PROGRAM FadenzugmotorAnAus
VAR
	PowerFadenzugmotor: MC_Power;
	PowerFadenzugmotorOut: ST_McOutputs;
	ResetFadenzugmotor: MC_Reset;
	ResetFadenzugmotorOut: ST_McOutputs;
	HaltFadenzugmotor: MC_Halt;
	HaltFadenzugmotorOut: ST_McOutputs;
	HomeFadenzugmotor: MC_Home;
	HomeFadenzugmotorOut: ST_McOutputs;
	MoveAbFadenzugmotorOut1: ST_McOutputs;
	MoveAbFadenzugmotor1: MC_MoveAbsolute;
	MoveAbFadenzugmotor2: MC_MoveAbsolute;
	MoveAbFadenzugmotorOut2: ST_McOutputs;
	MC_Stop1: MC_Stop;
	MC_StopOut1: ST_McOutputs;
	HaltAufwicklerOut: ST_McOutputs;
	HaltAbwicklerOut: ST_McOutputs;
	AbwicklerMoveV_Out: ST_McOutputs;
	AufwicklerMoveV: MC_MoveVelocity;
	HaltAbwickler: MC_Halt;
	HaltAufwickler: MC_Halt;
	PowerAbwickler: MC_Power;
	PowerAbwicklerOut: ST_McOutputs;
	PowerAufwickler: MC_Power;
	PowerAufwicklerOut: ST_McOutputs;
	HomeAbwickler: MC_Home;
	HomeAbwicklerOut: ST_McOutputs;
	HomeAufwickler: MC_Home;
	HomeAufwicklerOut: ST_McOutputs;
	ResetAbwickler: MC_Reset;
	ResetAbwickleOUT: ST_McOutputs;
	ResetAufwickler: MC_Reset;
	ResetAufwickleOUT: ST_McOutputs;
	MasterMoveV: MC_MoveVelocity;
	HaltMasterachse: MC_Halt;
	ResetMasterachseOut: ST_McOutputs;
	HomeMasterachseOut: ST_McOutputs;
	HaltMasterachseOut: ST_McOutputs;
	PowerMasterachseOut: ST_McOutputs;
	GearIn_M_AB_Out: ST_McOutputs;
	MasterMoveV_Out: ST_McOutputs;
	PowerMasterachse: MC_Power;
	HomeMasterachse: MC_Home;
	ResetMasterachse: MC_Reset;
	GearIn_M_AB: MC_GearIn;
	GearOut_M_AB: MC_GearOut;
	CamIn_AB_AUF_Out: ST_McOutputs;
	GearOut_M_AB_Out: ST_McOutputs;
	CamIn_AB_AUF: MC_CamIn;
	CamOut_AB_AUF: MC_CamOut;
	JogFadenzugmotorOut: ST_McOutputs;
	CamOut_AB_AUF_Out: ST_McOutputs;
	startFadenzugTrig: R_TRIG;
	flag: INT;
	JogFadenzugmotor: MC_Jog;
	// Zustandsvariable Hauptprogramm
	stateFadenzugmotor: MoveState_Fadenzugmotor;
	
END_VAR

GlobaleVariablen.Fadenzugmotor();
IF Fadenzugmotor.NcToPlc.ActPos > 89 AND Fadenzugmotor.NcToPlc.ActPos < 91 THEN
	FadenzugHomingFertig := TRUE;
ELSE FadenzugHomingFertig := FALSE;
END_IF
IF DTD_CTD THEN
	TrackingDifferentiator(Sollkraft);
ELSE
	DiscreteTrackingDifferentiator(Sollkraft);
END_IF

ESO(Fadenzugkraft_2);

// Programmablauf mittels Zustandsautomat
CASE stateFadenzugmotor OF
(* ===========================================================================================
	Zustand 1: Programm ist im Ausgangszustand und wartet auf Benutzereingabe. Alle 
	Funktionsbausteine werden initialisiert, etwaige Fehler zurückgesetzt. *)	
	FADENZUG_INIT:
		FadenzugmotorStopp := FALSE;
		MoveAbFadenzugmotor1.Execute := FALSE;
		MoveAbFadenzugmotor2.Execute := FALSE;
		FadenzugmotorLaeuft := FALSE;
		ResetFadenzugmotor.Execute := FALSE;
		HaltFadenzugmotor.Execute := FALSE;
		FadenmotorRegeln := FALSE;
		IF FadenmotorFreigabe THEN
			stateFadenzugmotor := FADENZUG_POWER_ON;
		ELSE
			PowerFadenzugmotor.Enable := FALSE;
			PowerFadenzugmotor.Enable_Positive := FALSE;
			PowerFadenzugmotor.Enable_Negative := FALSE;
		END_IF
(* ===========================================================================================
	Zustand 2: Schlalten der allgemeinen Software-Freigabe, Vorschubfreigabe in positive Richtung
	durch MC_Power. Sobald Funktionsbaustein MC_Power die Betriebsbereitschaft der Achse signalisiert,
	Zustandsübergang in Forward*)
	FADENZUG_POWER_ON:
		IF FadenmotorFreigabe = TRUE THEN
			PowerFadenzugmotor.Enable := TRUE;
			PowerFadenzugmotor.Enable_Positive := TRUE;
			PowerFadenzugmotor.Enable_Negative := TRUE;
			FadenzugmotorStopp := FALSE;
			IF PowerFadenzugmotorOut.Done THEN
				IF FadenzugJogStart THEN
					stateFadenzugmotor := FADENZUG_JOG;
				END_IF
			ELSIF PowerFadenzugmotor.Error THEN
				stateFadenzugmotor := FADENZUG_ERROR;
			END_IF
		ELSIF FadenmotorFreigabe = FALSE THEN
			stateFadenzugmotor := FADENZUG_HALT_ZU_INT;
		END_IF
(* ===========================================================================================
	Zustand 3: Setzten der Ist-Position auf 90 Grad*)			
	FADENZUG_JOG:
		IF FadenmotorFreigabe = TRUE THEN
			FadenzugmotorJogLaeuft := TRUE;
			ActJog();
			IF FadenzugJogStart = FALSE THEN
				FadenzugmotorJogLaeuft := FALSE;
				IF FadenmotorRegeln = TRUE THEN
					stateFadenzugmotor := FADENZUG_MOVE;
				END_IF
			END_IF
		ELSIF FadenmotorFreigabe = FALSE THEN
			stateFadenzugmotor := FADENZUG_HALT_ZU_INT;
		END_IF
(* ===========================================================================================
	Zustand 4: Starten des Fadenzugmotors mithilfe der Fadenzugspannung. Zustandsübergang durch Bedienerbefehl.*)	
	FADENZUG_MOVE:
	
		IF FadenmotorFreigabe = TRUE THEN
			
			IF FadenzugmotorStopp = TRUE THEN
				FadenmotorFreigabe := FALSE;
			END_IF
			//*********Positionsführungsgröße berechnen*************
			PRG_PID_Fadenzugmotor();
			IF ILC_EinAus = TRUE AND MasterStart = TRUE THEN
				ILC();
				MoveAbFadenzugmotor1.Position := ILC_Out + GlobaleVariablen.Fadenzugmotor.NcToPlc.ActPos + _u;
			ELSE
				MoveAbFadenzugmotor1.Position := GlobaleVariablen.Fadenzugmotor.NcToPlc.ActPos + _u;
			END_IF
			
			MoveAbFadenzugmotor1.Velocity := 60000;
			ActBegrenzung_1();
			//******************************************************
			
			MoveAbFadenzugmotor1.Execute := TRUE;
			FadenzugmotorLaeuft := TRUE;
			
			//*********Zustand umschalten***************************
			IF MoveAbFadenzugmotorOut1.Busy OR MoveAbFadenzugmotorOut1.Active THEN
				MoveAbFadenzugmotor1.Execute := FALSE;
				stateFadenzugmotor := FADENZUG_MOVE_NEW;
			END_IF
			
			IF MoveAbFadenzugmotorOut1.Done OR MoveAbFadenzugmotorOut1.CommandAborted THEN
				MoveAbFadenzugmotor1.Execute := FALSE;
				stateFadenzugmotor := FADENZUG_MOVE;
			END_IF

			IF MoveAbFadenzugmotorOut1.Error THEN
				stateFadenzugmotor := FADENZUG_ERROR;
			END_IF
			//******************************************************
		ELSIF FadenmotorFreigabe = FALSE THEN
			stateFadenzugmotor := FADENZUG_HALT_ZU_INT;
		END_IF
(* ===========================================================================================		
	Zustand 5: Die Funktion ist gleich wie Zustand 4, aber mithilfe dises Zustands kann den letzte Positionsbefehel unterbrechen 
	und schnell den neue Positionsbefehel aktualisieret und ersetzt werden. *)		
	FADENZUG_MOVE_NEW:

		IF FadenmotorFreigabe = TRUE THEN
			
			IF FadenzugmotorStopp = TRUE THEN
				FadenmotorFreigabe := FALSE;
			END_IF
			
			//*********Positionsführungsgröße berechnen*************
			PRG_PID_Fadenzugmotor();
			IF ILC_EinAus = TRUE AND MasterStart = TRUE THEN
				ILC();
				MoveAbFadenzugmotor2.Position := ILC_Out + GlobaleVariablen.Fadenzugmotor.NcToPlc.ActPos + _u;
			ELSE
				MoveAbFadenzugmotor2.Position := GlobaleVariablen.Fadenzugmotor.NcToPlc.ActPos + _u;
			END_IF
			MoveAbFadenzugmotor2.Velocity := 60000;
			ActBegrenzung_2();
			//******************************************************
			
			MoveAbFadenzugmotor2.Execute := TRUE;
			FadenzugmotorLaeuft := TRUE;
			
			//*********Zustand umschalten***************************
			IF MoveAbFadenzugmotorOut2.Busy OR MoveAbFadenzugmotorOut2.Active THEN
				MoveAbFadenzugmotor2.Execute := FALSE;
				stateFadenzugmotor := FADENZUG_MOVE;
			ELSIF MoveAbFadenzugmotorOut2.Done OR MoveAbFadenzugmotorOut2.CommandAborted THEN
				MoveAbFadenzugmotor2.Execute := FALSE;
				stateFadenzugmotor := FADENZUG_MOVE_NEW;
			ELSIF MoveAbFadenzugmotorOut2.Error THEN
				stateFadenzugmotor := FADENZUG_ERROR;
			END_IF
			//******************************************************
		ELSIF FadenmotorFreigabe = FALSE THEN
			stateFadenzugmotor := FADENZUG_HALT_ZU_INT;
		END_IF
(* ===========================================================================================
   Zustand 7: Anhalten des Fadenzugmotors, im Anschluss Rückkehr in den Ausgangszustand. *)			
	FADENZUG_HALT_ZU_INT:
		MoveAbFadenzugmotor1.Execute := FALSE;
		MoveAbFadenzugmotor2.Execute := FALSE;
		HaltFadenzugmotor.Execute := TRUE;
		IF HaltFadenzugmotorOut.Done THEN
			FadenzugmotorStopp := TRUE;
			FadenmotorFreigabe := FALSE;
			FadenzugmotorLaeuft := FALSE;
			HaltFadenzugmotor.Execute := FALSE;
			stateFadenzugmotor := FADENZUG_INIT;
		ELSIF HaltFadenzugmotorOut.Error OR HaltFadenzugmotorOut.CommandAborted THEN
			HaltFadenzugmotor.Execute := FALSE;
			stateFadenzugmotor := FADENZUG_ERROR;
		END_IF

(* ===========================================================================================
   Zustand 8: Im Falle eines Bausteinfehlers wird überprüft, ob sich die Achse ebenfalls im    
   Fehlerzustand befindet, was einen Achsreset erfordert. Andernfalls werden Bausteinfehler 
   im Zustand Init zurückgesetzt.*)				
	FADENZUG_ERROR:
		MoveAbFadenzugmotor1.Execute := FALSE;
		MoveAbFadenzugmotor2.Execute := FALSE;
		PowerFadenzugmotor.Enable := FALSE;
		FadenmotorFreigabe := FALSE;
		IF Fadenzugmotor.Status.Error THEN
			stateFadenzugmotor := FADENZUG_RESET;	// Reset bei Achsfehler
		ELSE
			stateFadenzugmotor := FADENZUG_INIT;	// Funktionsbausteinfehler erfordert keinen Reset
		END_IF
(* ===========================================================================================
   Zustand 9:  Durchführung des Achsreset im Fehlerfall  *)	
	FADENZUG_RESET:
		MoveAbFadenzugmotor1.Execute := FALSE;
		MoveAbFadenzugmotor2.Execute := FALSE;
		PowerFadenzugmotor.Enable := FALSE;
		ResetFadenzugmotor.Execute := TRUE;
		FadenmotorFreigabe := FALSE;
		IF ResetFadenzugmotor.Done THEN
			FadenzugmotorLaeuft := FALSE;
			stateFadenzugmotor := FADENZUG_INIT;
		ELSIF ResetFadenzugmotorOut.Error THEN
			stateFadenzugmotor := FADENZUG_INIT; (* Falls Reset nicht gelingt, Benutzereingriff erforderlich *)
		END_IF
END_CASE

// Zyklusmäßige Aufrufe
ActPower();		// Aufruf des Funktionsbausteines
ActHalt();
ActRest();
ActMoveAbsolute();

ACTION ActBegrenzung_1:

IF FadenzugmotorAnAus.MoveAbFadenzugmotor1.Position > MaxPosition THEN
	MoveAbFadenzugmotor1.Position := MaxPosition;
	MoveAbFadenzugmotor1.Velocity := 100;
ELSIF FadenzugmotorAnAus.MoveAbFadenzugmotor1.Position < MinPosition THEN
	MoveAbFadenzugmotor1.Position := MinPosition;
	MoveAbFadenzugmotor1.Velocity := 100;
END_IF

IF Fadenzugmotor.NcToPlc.ActPos < MinPosition THEN
	MoveAbFadenzugmotor1.Position := MinPosition;
	MoveAbFadenzugmotor1.Velocity := 100;
	MoveAbFadenzugmotor1.Execute := TRUE;
ELSIF Fadenzugmotor.NcToPlc.ActPos > MaxPosition THEN
	MoveAbFadenzugmotor1.Position := MaxPosition;
	MoveAbFadenzugmotor1.Velocity := 100;
	MoveAbFadenzugmotor1.Execute := TRUE;
END_IF
END_ACTION

ACTION ActBegrenzung_2:
IF MoveAbFadenzugmotor2.Position > MaxPosition THEN
MoveAbFadenzugmotor2.Position := MaxPosition;
MoveAbFadenzugmotor2.Velocity := 100;
ELSIF MoveAbFadenzugmotor2.Position < MinPosition THEN
	MoveAbFadenzugmotor2.Position := MinPosition;
	MoveAbFadenzugmotor2.Velocity := 100;
END_IF

IF Fadenzugmotor.NcToPlc.ActPos < MinPosition THEN
	MoveAbFadenzugmotor2.Position := MinPosition;
	MoveAbFadenzugmotor2.Velocity := 100;
	MoveAbFadenzugmotor2.Execute := TRUE;
ELSIF Fadenzugmotor.NcToPlc.ActPos > MaxPosition THEN
	MoveAbFadenzugmotor2.Position := MaxPosition;
	MoveAbFadenzugmotor2.Velocity := 100;
	MoveAbFadenzugmotor2.Execute := TRUE;
END_IF
END_ACTION

ACTION ActHalt:
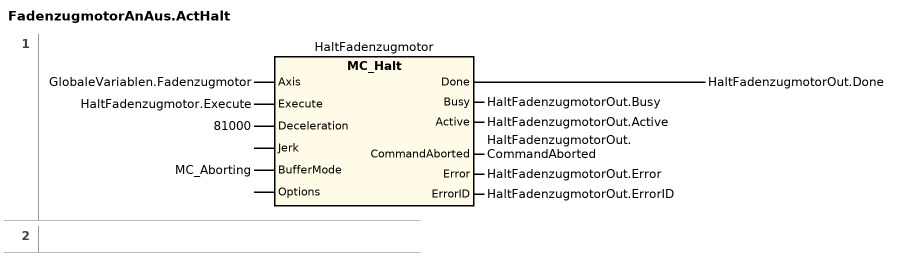
// NETWORK 1
HaltFadenzugmotor(
    Axis := GlobaleVariablen.Fadenzugmotor,
    Execute := HaltFadenzugmotor.Execute,
    Deceleration := 81000,
    BufferMode := MC_Aborting,
    Busy => HaltFadenzugmotorOut.Busy,
    Active => HaltFadenzugmotorOut.Active,
    CommandAborted => HaltFadenzugmotorOut.CommandAborted,
    Error => HaltFadenzugmotorOut.Error,
    ErrorID => HaltFadenzugmotorOut.ErrorID); // MC_Halt
HaltFadenzugmotorOut.Done := HaltFadenzugmotor.Done;

// NETWORK 2
END_ACTION

ACTION ActJog:
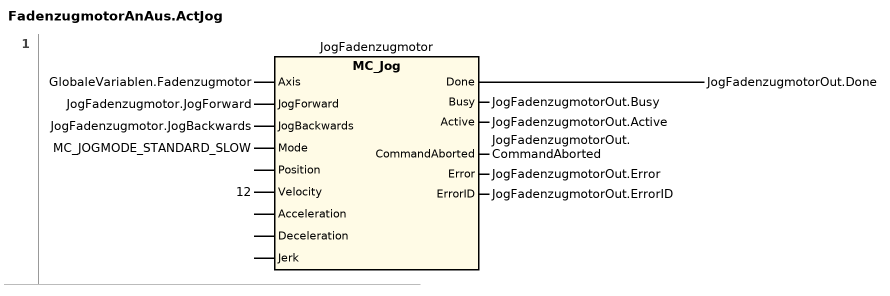
// NETWORK 1
JogFadenzugmotor(
    Axis := GlobaleVariablen.Fadenzugmotor,
    JogForward := JogFadenzugmotor.JogForward,
    JogBackwards := JogFadenzugmotor.JogBackwards,
    Mode := MC_JOGMODE_STANDARD_SLOW,
    Velocity := 12,
    Busy => JogFadenzugmotorOut.Busy,
    Active => JogFadenzugmotorOut.Active,
    CommandAborted => JogFadenzugmotorOut.CommandAborted,
    Error => JogFadenzugmotorOut.Error,
    ErrorID => JogFadenzugmotorOut.ErrorID); // MC_Jog
JogFadenzugmotorOut.Done := JogFadenzugmotor.Done;
END_ACTION

ACTION ActMoveAbsolute:
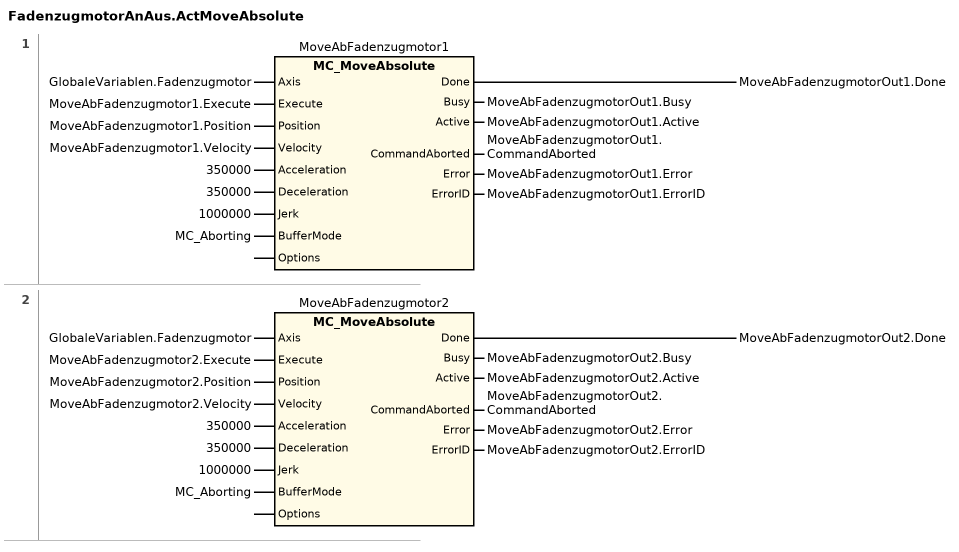
// NETWORK 1
MoveAbFadenzugmotor1(
    Axis := GlobaleVariablen.Fadenzugmotor,
    Execute := MoveAbFadenzugmotor1.Execute,
    Position := MoveAbFadenzugmotor1.Position,
    Velocity := MoveAbFadenzugmotor1.Velocity,
    Acceleration := 350000,
    Deceleration := 350000,
    Jerk := 1000000,
    BufferMode := MC_Aborting,
    Busy => MoveAbFadenzugmotorOut1.Busy,
    Active => MoveAbFadenzugmotorOut1.Active,
    CommandAborted => MoveAbFadenzugmotorOut1.CommandAborted,
    Error => MoveAbFadenzugmotorOut1.Error,
    ErrorID => MoveAbFadenzugmotorOut1.ErrorID); // MC_MoveAbsolute
MoveAbFadenzugmotorOut1.Done := MoveAbFadenzugmotor1.Done;

// NETWORK 2
MoveAbFadenzugmotor2(
    Axis := GlobaleVariablen.Fadenzugmotor,
    Execute := MoveAbFadenzugmotor2.Execute,
    Position := MoveAbFadenzugmotor2.Position,
    Velocity := MoveAbFadenzugmotor2.Velocity,
    Acceleration := 350000,
    Deceleration := 350000,
    Jerk := 1000000,
    BufferMode := MC_Aborting,
    Busy => MoveAbFadenzugmotorOut2.Busy,
    Active => MoveAbFadenzugmotorOut2.Active,
    CommandAborted => MoveAbFadenzugmotorOut2.CommandAborted,
    Error => MoveAbFadenzugmotorOut2.Error,
    ErrorID => MoveAbFadenzugmotorOut2.ErrorID); // MC_MoveAbsolute
MoveAbFadenzugmotorOut2.Done := MoveAbFadenzugmotor2.Done;
END_ACTION

ACTION ActPower:
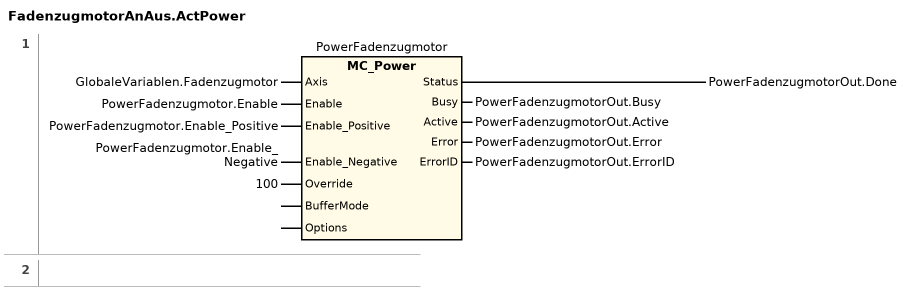
// NETWORK 1
PowerFadenzugmotor(
    Axis := GlobaleVariablen.Fadenzugmotor,
    Enable := PowerFadenzugmotor.Enable,
    Enable_Positive := PowerFadenzugmotor.Enable_Positive,
    Enable_Negative := PowerFadenzugmotor.Enable_Negative,
    Override := 100,
    Busy => PowerFadenzugmotorOut.Busy,
    Active => PowerFadenzugmotorOut.Active,
    Error => PowerFadenzugmotorOut.Error,
    ErrorID => PowerFadenzugmotorOut.ErrorID); // MC_Power
PowerFadenzugmotorOut.Done := PowerFadenzugmotor.Status;

// NETWORK 2
END_ACTION

ACTION ActRest:
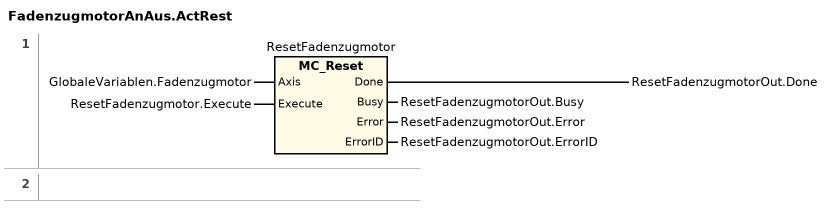
// NETWORK 1
ResetFadenzugmotor(
    Axis := GlobaleVariablen.Fadenzugmotor,
    Execute := ResetFadenzugmotor.Execute,
    Busy => ResetFadenzugmotorOut.Busy,
    Error => ResetFadenzugmotorOut.Error,
    ErrorID => ResetFadenzugmotorOut.ErrorID); // MC_Reset
ResetFadenzugmotorOut.Done := ResetFadenzugmotor.Done;

// NETWORK 2
END_ACTION

END_PROGRAM

(* stored: Version 1.1.0.1, ProductVersion 3.1.4024.11
   POU FadenzugmotorAnAus: Id {a80a1380-31ec-4f5b-88df-eeb6854b3cea}, SpecialFunc None
   Action ActBegrenzung_1: Id {8103b026-4d45-43a3-907b-001a55e2b668}
   Action ActBegrenzung_2: Id {4188ac8d-43c1-4700-98a3-3591f3ae79b9}
   Action ActHalt: Id {b167bf1b-4469-430d-8ffc-f8df360ac471}
   Action ActJog: Id {b5a5e28e-ce30-4794-8f6d-abe3ccaac327}
   Action ActMoveAbsolute: Id {28c58b15-4e54-4828-b9c8-c363844d604c}
   Action ActPower: Id {b00ce2f7-9d11-479c-8b4d-c9643a1e206b}
   Action ActRest: Id {ac0bfe8b-9c78-46d3-b104-8ae3e6ca35ec} *)
